FUNCTION_BLOCK FB_EVENT_LISTENER
VAR_INPUT
	refFbEventFilter  : REFERENCE TO FB_TcEventFilter; 
	refFbTime:  REFERENCE TO FB_TIME;
END_VAR
VAR_OUTPUT
END_VAR
VAR
	hr : HRESULT;
	
	bSubscribe : BOOL := TRUE;
	bSubscribed : BOOL;
	bUnSubscribe : BOOL;
	
	fbMessageListener : FB_SAMPLE_LISTENER;
	Message: INT;
	
END_VAR

fbMessageListener.CustomExecute(refFbTime); // retrieve messages and its texts


IF bSubscribe THEN 
	bSubscribe := FALSE;
	hr := fbMessageListener.Subscribe2(refFbEventFilter); //subscribe to retrieve defined events
	IF SUCCEEDED(hr) THEN	
		bSubscribed := TRUE;
	END_IF
END_IF 

IF bUnSubscribe THEN 
	bUnSubscribe := FALSE;
	hr := fbMessageListener.Unsubscribe();
	IF SUCCEEDED(hr) THEN	
		bSubscribed := FALSE;
	END_IF
END_IF

END_FUNCTION_BLOCK

(* stored: Version 1.1.0.1, ProductVersion 3.1.4024.11
   POU FB_EVENT_LISTENER: Id {3f56ea05-5d12-4cf3-aa32-b1078ff3baf8}, SpecialFunc None *)
